// TIA Portal V18 export
FUNCTION_BLOCK "mot_universal_arrived_missed"   // FB70, FBD
{ S7_Optimized_Access := 'TRUE' }
VERSION : 0.1
// stored: AutoNumber true, IsIECCheckEnabled false, IsRetainMemResEnabled false, MemoryReserve 100, SetENOAutomatically false, UDAEnableTagReadback false
   VAR_INPUT
      target : Real;
      pos : Real;
   END_VAR
   VAR_OUTPUT
      arrived_misesd : Bool;
   END_VAR
   VAR
      target_was : Real;
      dir_to_target_pos : Bool;
      dir_to_target_pos_was : Bool;
   END_VAR
BEGIN

REGION Network 2 (SCL)
   #dir_to_target_pos := #pos < #target;

   IF #target = #target_was THEN
       #arrived_misesd := #dir_to_target_pos XOR #dir_to_target_pos_was;
   ELSE
       #arrived_misesd := false;

   END_IF;

   #target_was := #target;
   #dir_to_target_pos_was := #dir_to_target_pos;
END_REGION
END_FUNCTION_BLOCK
